(* IEC 61131-3 sources: ATCMcontrol_Engineering/src/COM/softing/fc/AddOns/Softing/4CPCTarget/Libs/ATCM_IEC1131_3/table_25, 4 files *)

(* ---- rol.st ---- *)
(*[[
    UserURL= "ATCM:ROL.htm"
]]*)

FUNCTION ROL : ANY_BIT
VAR_INPUT
    IN : ANY_BIT;
    N  : ANY_INT;
END_VAR

overload BOOL(BOOL,DINT)   inline{%1}
overload BYTE(BYTE,DINT)   inline{Utils.rol(%1,%2,8)}
overload WORD(WORD,DINT)   inline{Utils.rol(%1,%2,16)}
overload DWORD(DWORD,DINT) inline{Utils.rol(%1,%2,32)}
overload LWORD(LWORD,DINT) inline{Utils.rol_l(%1,%2)}

END_FUNCTION

(* ---- ror.st ---- *)
(*[[
    UserURL= "ATCM:ROR.htm"
]]*)

FUNCTION ROR : ANY_BIT
VAR_INPUT
    IN : ANY_BIT;
    N  : ANY_INT;
END_VAR

overload BOOL(BOOL,DINT)   inline{%1}
overload BYTE(BYTE,DINT)   inline{Utils.ror(%1,%2,8)}
overload WORD(WORD,DINT)   inline{Utils.ror(%1,%2,16)}
overload DWORD(DWORD,DINT) inline{Utils.ror(%1,%2,32)}
overload LWORD(LWORD,DINT) inline{Utils.ror_l(%1,%2)}

END_FUNCTION

(* ---- shl.st ---- *)
(*[[
    UserURL= "ATCM:SHL.htm"
]]*)

FUNCTION SHL : ANY_BIT
VAR_INPUT
    IN : ANY_BIT;
    N  : ANY_INT;
END_VAR

overload BOOL(BOOL,DINT)   inline{Utils.shift_bool(%1,%2)}
overload BYTE(BYTE,DINT)   inline{Utils.shl(%1,%2,8)}
overload WORD(WORD,DINT)   inline{Utils.shl(%1,%2,16)}
overload DWORD(DWORD,DINT) inline{Utils.shl(%1,%2,32)}
overload LWORD(LWORD,DINT) inline{Utils.shl_l(%1,%2)}

END_FUNCTION

(* ---- shr.st ---- *)
(*[[
    UserURL= "ATCM:SHR.htm"
]]*)

FUNCTION SHR : ANY_BIT
VAR_INPUT
    IN : ANY_BIT;
    N  : ANY_INT;
END_VAR

overload BOOL (BOOL, DINT)   inline{Utils.shift_bool(%1,%2)}
overload BYTE (BYTE, DINT)   inline{Utils.shr(%1,%2,8)}
overload WORD (WORD, DINT)   inline{Utils.shr(%1,%2,16)}
overload DWORD(DWORD,DINT)   inline{Utils.shr(%1,%2,32)}
overload LWORD(LWORD,DINT)   inline{Utils.shr_l(%1,%2)}

END_FUNCTION
